(* IEC 61131-3 sources: controlforge-structured-text/iec61131-definitions, 10 files *)

(* ---- CTD.st ---- *)
(*
    CTD - Count Down Counter (IEC 61131-3)

    CV decrements by 1 on each rising edge of CD.
    Q becomes TRUE when CV <= 0.
    LD loads PV into CV when TRUE.

    Typical uses: remaining inventory, countdown sequences, quota tracking.

    Example:
        Countdown(CD := ItemDispensed, LD := Reload, PV := 50);
        IF Countdown.Q THEN
            // All items dispensed
        END_IF;
*)

FUNCTION_BLOCK CTD
VAR_INPUT
    CD : BOOL;      // Count down - CV decrements on rising edge
    LD : BOOL;      // Load - sets CV to PV when TRUE
    PV : INT;       // Preset value - initial count loaded by LD
END_VAR
VAR_OUTPUT
    Q : BOOL;       // Output - TRUE when CV <= 0
    CV : INT;       // Current value - running count
END_VAR

END_FUNCTION_BLOCK

(* ---- CTU.st ---- *)
(*
    CTU - Count Up Counter (IEC 61131-3)

    CV increments by 1 on each rising edge of CU.
    Q becomes TRUE when CV >= PV.
    R resets CV to 0 and Q to FALSE.

    Typical uses: production counting, cycle tracking, batch quantities.

    Example:
        Counter(CU := PartSensor, R := ResetBtn, PV := 100);
        IF Counter.Q THEN
            // 100 parts counted
        END_IF;
*)

FUNCTION_BLOCK CTU
VAR_INPUT
    CU : BOOL;      // Count up - CV increments on rising edge
    R : BOOL;       // Reset - sets CV to 0 when TRUE
    PV : INT;       // Preset value - target count for Q output
END_VAR
VAR_OUTPUT
    Q : BOOL;       // Output - TRUE when CV >= PV
    CV : INT;       // Current value - running count
END_VAR

END_FUNCTION_BLOCK

(* ---- CTUD.st ---- *)
(*
    CTUD - Count Up/Down Counter (IEC 61131-3)

    CV increments on rising edge of CU, decrements on rising edge of CD.
    QU becomes TRUE when CV >= PV.
    QD becomes TRUE when CV <= 0.
    R resets CV to 0. LD loads PV into CV.

    Typical uses: position tracking, bidirectional counting, balance calculations.

    Example:
        BiCounter(CU := AddPart, CD := RemovePart, R := FALSE, LD := FALSE, PV := 100);
        IF BiCounter.QU THEN
            // Upper limit reached
        END_IF;
*)

FUNCTION_BLOCK CTUD
VAR_INPUT
    CU : BOOL;      // Count up - CV increments on rising edge
    CD : BOOL;      // Count down - CV decrements on rising edge
    R : BOOL;       // Reset - sets CV to 0 when TRUE
    LD : BOOL;      // Load - sets CV to PV when TRUE
    PV : INT;       // Preset value - target for QU, load value for LD
END_VAR
VAR_OUTPUT
    QU : BOOL;      // Up output - TRUE when CV >= PV
    QD : BOOL;      // Down output - TRUE when CV <= 0
    CV : INT;       // Current value - running count
END_VAR

END_FUNCTION_BLOCK

(* ---- F_TRIG.st ---- *)
(*
    F_TRIG - Falling Edge Detector (IEC 61131-3)

    Q is TRUE for exactly one scan cycle when CLK transitions TRUE -> FALSE.
    Q is FALSE at all other times.
    Uses internal memory M to track previous CLK state.

    Typical uses: stop command detection, end-of-cycle detection, falling alarm acknowledgment.

    Example:
        StopEdge(CLK := RunningSignal);
        IF StopEdge.Q THEN
            // Signal just dropped (one-shot)
        END_IF;
*)

FUNCTION_BLOCK F_TRIG
VAR_INPUT
    CLK : BOOL;     // Clock input - signal to monitor for falling edge
END_VAR
VAR_OUTPUT
    Q : BOOL;       // Output - TRUE for one scan on TRUE->FALSE transition
END_VAR
VAR
    M : BOOL;       // Internal memory - previous CLK state
END_VAR

END_FUNCTION_BLOCK

(* ---- R_TRIG.st ---- *)
(*
    R_TRIG - Rising Edge Detector (IEC 61131-3)

    Q is TRUE for exactly one scan cycle when CLK transitions FALSE -> TRUE.
    Q is FALSE at all other times.
    Uses internal memory M to track previous CLK state.

    Typical uses: button press detection, start triggers, rising alarm conditions.

    Example:
        StartEdge(CLK := StartButton);
        IF StartEdge.Q THEN
            // Start button just pressed (one-shot)
        END_IF;
*)

FUNCTION_BLOCK R_TRIG
VAR_INPUT
    CLK : BOOL;     // Clock input - signal to monitor for rising edge
END_VAR
VAR_OUTPUT
    Q : BOOL;       // Output - TRUE for one scan on FALSE->TRUE transition
END_VAR
VAR
    M : BOOL;       // Internal memory - previous CLK state
END_VAR

END_FUNCTION_BLOCK

(* ---- RS.st ---- *)
(*
    RS - Reset-Dominant Bistable (IEC 61131-3)

    Latching flip-flop where reset (R1) has priority over set (S).
    Q1 = TRUE when S is TRUE and R1 is FALSE.
    Q1 = FALSE when R1 is TRUE (regardless of S).
    Q1 holds state when both S and R1 are FALSE.

    Typical uses: emergency stop latches, fault conditions requiring manual reset.

    Example:
        EStopLatch(S := StartPermit, R1 := EStopPressed);
        MotorEnable := EStopLatch.Q1;
        // EStop always overrides start permit
*)

FUNCTION_BLOCK RS
VAR_INPUT
    S : BOOL;       // Set input - sets Q1 TRUE (non-dominant)
    R1 : BOOL;      // Reset input - resets Q1 FALSE (dominant, priority)
END_VAR
VAR_OUTPUT
    Q1 : BOOL;      // Output - latched bistable state
END_VAR

END_FUNCTION_BLOCK

(* ---- SR.st ---- *)
(*
    SR - Set-Dominant Bistable (IEC 61131-3)

    Latching flip-flop where set (S1) has priority over reset (R).
    Q1 = TRUE when S1 is TRUE (regardless of R).
    Q1 = FALSE when R is TRUE and S1 is FALSE.
    Q1 holds state when both S1 and R are FALSE.

    Typical uses: start/run conditions, permissive latches.

    Example:
        RunLatch(S1 := StartCmd, R := StopCmd);
        Running := RunLatch.Q1;
        // Start always overrides stop
*)

FUNCTION_BLOCK SR
VAR_INPUT
    S1 : BOOL;      // Set input - sets Q1 TRUE (dominant, priority)
    R : BOOL;       // Reset input - resets Q1 FALSE (non-dominant)
END_VAR
VAR_OUTPUT
    Q1 : BOOL;      // Output - latched bistable state
END_VAR

END_FUNCTION_BLOCK

(* ---- TOF.st ---- *)
(*
    TOF - Off-Delay Timer (IEC 61131-3)

    Q is TRUE while IN is TRUE. When IN goes FALSE, timer starts.
    Q stays TRUE until ET reaches PT, then Q goes FALSE.
    If IN goes TRUE again before PT, timer resets.

    Typical uses: cooling fan run-on, valve close delays, shutdown sequences.

    Example:
        FanDelay(IN := MotorRunning, PT := T#30s);
        FanOutput := FanDelay.Q;
        // Fan stays on 30s after motor stops
*)

FUNCTION_BLOCK TOF
VAR_INPUT
    IN : BOOL;      // Timer input - Q follows IN while TRUE
    PT : TIME;      // Preset time - off-delay duration after IN goes FALSE
END_VAR
VAR_OUTPUT
    Q : BOOL;       // Output - TRUE while IN is TRUE or timer running
    ET : TIME;      // Elapsed time - counts from T#0s to PT after IN goes FALSE
END_VAR

END_FUNCTION_BLOCK

(* ---- TON.st ---- *)
(*
    TON - On-Delay Timer (IEC 61131-3)

    Starts timing when IN transitions FALSE -> TRUE.
    Q becomes TRUE after elapsed time ET reaches preset PT.
    Q stays TRUE while IN remains TRUE.
    When IN goes FALSE, Q resets immediately and ET resets to T#0s.

    Typical uses: motor start delays, alarm confirmation, process step durations.

    Example:
        MyTimer(IN := StartCondition, PT := T#5s);
        IF MyTimer.Q THEN
            // 5 seconds elapsed since StartCondition went TRUE
        END_IF;
*)

FUNCTION_BLOCK TON
VAR_INPUT
    IN : BOOL;      // Start signal - rising edge starts timer
    PT : TIME;      // Preset time - delay duration before Q goes TRUE
END_VAR
VAR_OUTPUT
    Q : BOOL;       // Output - TRUE when ET >= PT and IN is TRUE
    ET : TIME;      // Elapsed time - counts from T#0s to PT while IN is TRUE
END_VAR

END_FUNCTION_BLOCK

(* ---- TP.st ---- *)
(*
    TP - Pulse Timer (IEC 61131-3)

    Generates a fixed-duration pulse on rising edge of IN.
    Q goes TRUE immediately on IN rising edge and stays TRUE for PT.
    New rising edges during active pulse are ignored.
    ET counts up to PT then stops.

    Typical uses: momentary outputs, reset pulses, notification signals.

    Example:
        Pulse(IN := TriggerInput, PT := T#500ms);
        PulseOutput := Pulse.Q;
        // 500ms pulse on each rising edge of TriggerInput
*)

FUNCTION_BLOCK TP
VAR_INPUT
    IN : BOOL;      // Trigger input - rising edge starts pulse
    PT : TIME;      // Preset time - pulse duration
END_VAR
VAR_OUTPUT
    Q : BOOL;       // Pulse output - TRUE for duration PT
    ET : TIME;      // Elapsed time - counts from T#0s to PT during pulse
END_VAR

END_FUNCTION_BLOCK
